(* CoDeSys 2.3 export: TACT_BUTTON.EXP *)

(* POU 05_Basic_Calc/tact_button, CFC *)
FUNCTION_BLOCK tact_button
VAR_INPUT
	button:	BOOL;
END_VAR
VAR_OUTPUT
	state:	BOOL;
END_VAR
VAR
	rtr1:	R_TRIG;
	rs1: 	RS;
END_VAR
VAR (* helpers for the ST form of the networks *)
	_t254 : BOOL;
	_t258 : BOOL;
END_VAR
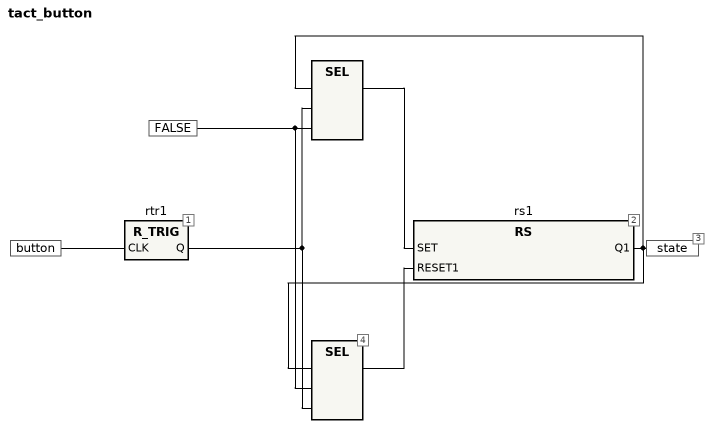
_CFC_ (* Continuous Function Chart, elements in execution order *)
#0 SEL(#2.Q1, #1.Q, FALSE)
#1 rtr1:R_TRIG(CLK: button)
#2 rs1:RS(SET: #0, RESET1: #4)
#3 state <= #2.Q1
#4 SEL(#2.Q1, FALSE, #1.Q)
_END_CFC_
(* the same logic as Structured Text *)
_t254 := SEL(rs1.Q1, rtr1.Q, FALSE);
rtr1(CLK := button);
rs1(SET := _t254, RESET1 := _t258);
state := rs1.Q1;
_t258 := SEL(rs1.Q1, FALSE, rtr1.Q);
END_FUNCTION_BLOCK
